// TIA Portal V17 export
// export: Created 2023-03-06T02:05:21.4493733Z, ExportSetting WithDefaults, DisplayName Totally Integrated Automation Portal, DisplayVersion V17 Update 4, DisplayName TIA Portal Openness, DisplayVersion V17 Update 4, DisplayName TIA Portal Version Control Interface, DisplayVersion V17, DisplayName STEP 7 Professional, DisplayVersion V17 Update 4, DisplayName STEP 7 Safety, DisplayVersion V17, DisplayName WinCC Professional, DisplayVersion V17 Update 4
FUNCTION "SM2_Logic" : Void   // FC70, LAD
TITLE = State Machine Logic
{ S7_Optimized_Access := 'TRUE' }
VERSION : 0.1
// stored: AutoNumber false, IsIECCheckEnabled false, SetENOAutomatically false, UDAEnableTagReadback false
   VAR_TEMP   // added for the SCL form of the ladder/FBD networks
      _w1 : Bool;
   END_VAR
BEGIN

REGION Network 1: Stop Command
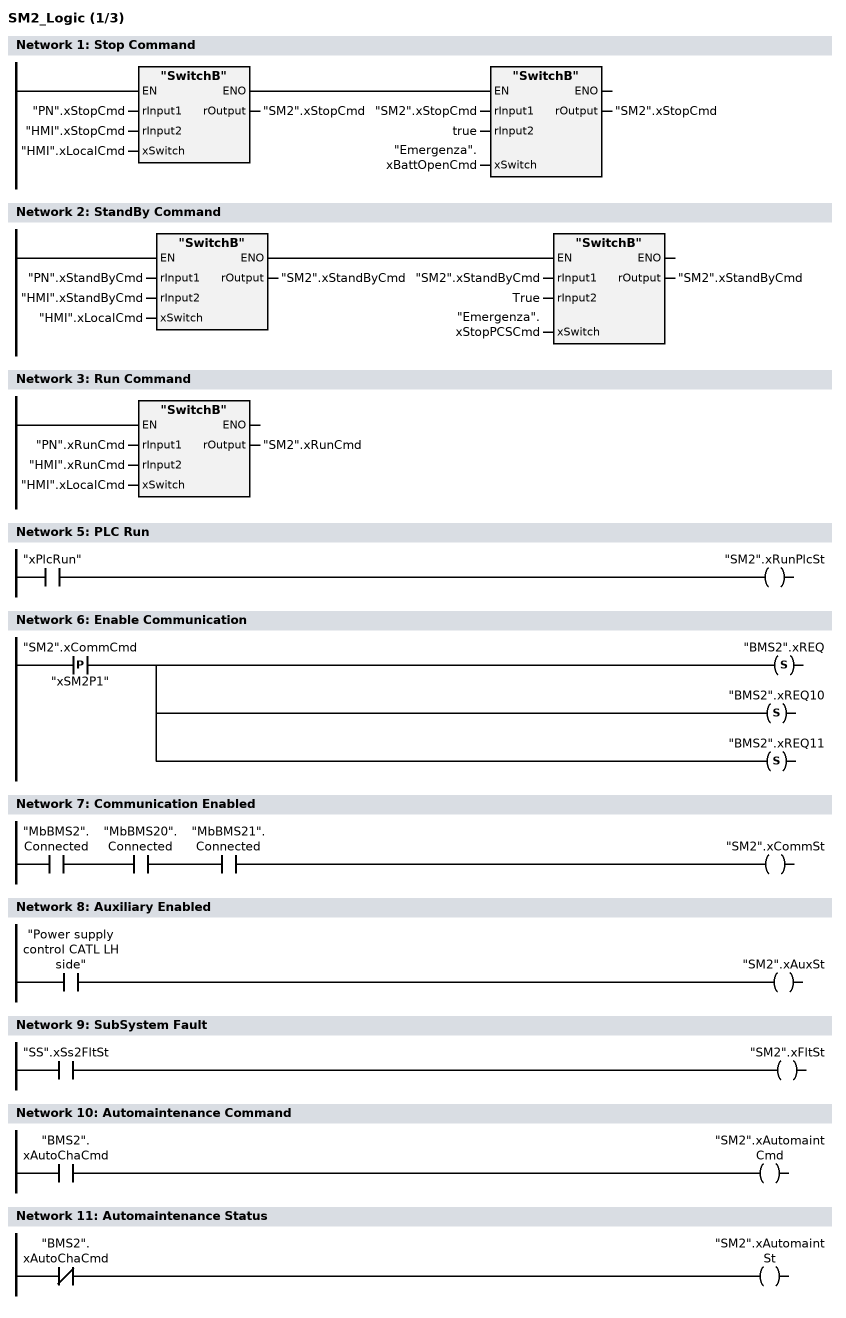
   RUNG wire#powerrail
      "SwitchB"(rInput1 := "PN".xStopCmd, rInput2 := "HMI".xStopCmd, xSwitch := "HMI".xLocalCmd, rOutput => "SM2".xStopCmd)
      "SwitchB"(rInput1 := "SM2".xStopCmd, rInput2 := true, xSwitch := "Emergenza".xBattOpenCmd, rOutput => "SM2".xStopCmd)
   END_RUNG
   // the same network as SCL:
   "SwitchB"(rInput1 := "PN".xStopCmd,
             rInput2 := "HMI".xStopCmd,
             xSwitch := "HMI".xLocalCmd,
             rOutput => "SM2".xStopCmd,
             ENO => #_w1);
   IF #_w1 THEN
       "SwitchB"(rInput1 := "SM2".xStopCmd,
                 rInput2 := true,
                 xSwitch := "Emergenza".xBattOpenCmd,
                 rOutput => "SM2".xStopCmd);
   END_IF;
END_REGION

REGION Network 2: StandBy Command
   RUNG wire#powerrail
      "SwitchB"(rInput1 := "PN".xStandByCmd, rInput2 := "HMI".xStandByCmd, xSwitch := "HMI".xLocalCmd, rOutput => "SM2".xStandByCmd)
      "SwitchB"(rInput1 := "SM2".xStandByCmd, rInput2 := True, xSwitch := "Emergenza".xStopPCSCmd, rOutput => "SM2".xStandByCmd)
   END_RUNG
   // the same network as SCL:
   "SwitchB"(rInput1 := "PN".xStandByCmd,
             rInput2 := "HMI".xStandByCmd,
             xSwitch := "HMI".xLocalCmd,
             rOutput => "SM2".xStandByCmd,
             ENO => #_w1);
   IF #_w1 THEN
       "SwitchB"(rInput1 := "SM2".xStandByCmd,
                 rInput2 := True,
                 xSwitch := "Emergenza".xStopPCSCmd,
                 rOutput => "SM2".xStandByCmd);
   END_IF;
END_REGION

REGION Network 3: Run Command
   RUNG wire#powerrail
      "SwitchB"(rInput1 := "PN".xRunCmd, rInput2 := "HMI".xRunCmd, xSwitch := "HMI".xLocalCmd, rOutput => "SM2".xRunCmd)
   END_RUNG
   // the same network as SCL:
   "SwitchB"(rInput1 := "PN".xRunCmd,
             rInput2 := "HMI".xRunCmd,
             xSwitch := "HMI".xLocalCmd,
             rOutput => "SM2".xRunCmd);
END_REGION

REGION Network 5: PLC Run
   RUNG wire#powerrail
      Contact( "xPlcRun" )
      Coil( "SM2".xRunPlcSt )
   END_RUNG
   // the same network as SCL:
   "SM2".xRunPlcSt := "xPlcRun";
END_REGION

REGION Network 6: Enable Communication
   RUNG wire#powerrail
      P_Contact(operand := "SM2".xCommCmd, bit := "xSM2P1")
      wire#w1
      S_Coil( "BMS2".xREQ )
   END_RUNG
   RUNG wire#w1
      S_Coil( "BMS2".xREQ10 )
   END_RUNG
   RUNG wire#w1
      S_Coil( "BMS2".xREQ11 )
   END_RUNG
   // the same network as SCL:
   #_w1 := "SM2".xCommCmd AND NOT "xSM2P1";   // rising edge of "SM2".xCommCmd
   "xSM2P1" := "SM2".xCommCmd;
   IF #_w1 THEN
       "BMS2".xREQ := TRUE;
       "BMS2".xREQ10 := TRUE;
       "BMS2".xREQ11 := TRUE;
   END_IF;
END_REGION

REGION Network 7: Communication Enabled
   RUNG wire#powerrail
      Contact( "MbBMS2".Connected )
      Contact( "MbBMS20".Connected )
      Contact( "MbBMS21".Connected )
      Coil( "SM2".xCommSt )
   END_RUNG
   // the same network as SCL:
   "SM2".xCommSt := "MbBMS2".Connected AND "MbBMS20".Connected AND "MbBMS21".Connected;
END_REGION

REGION Network 8: Auxiliary Enabled
   RUNG wire#powerrail
      Contact( "Power supply control CATL LH side" )
      Coil( "SM2".xAuxSt )
   END_RUNG
   // the same network as SCL:
   "SM2".xAuxSt := "Power supply control CATL LH side";
END_REGION

REGION Network 9: SubSystem Fault
   RUNG wire#powerrail
      Contact( "SS".xSs2FltSt )
      Coil( "SM2".xFltSt )
   END_RUNG
   // the same network as SCL:
   "SM2".xFltSt := "SS".xSs2FltSt;
END_REGION

REGION Network 10: Automaintenance Command
   RUNG wire#powerrail
      Contact( "BMS2".xAutoChaCmd )
      Coil( "SM2".xAutomaintCmd )
   END_RUNG
   // the same network as SCL:
   "SM2".xAutomaintCmd := "BMS2".xAutoChaCmd;
END_REGION

REGION Network 11: Automaintenance Status
   RUNG wire#powerrail
      I_Contact( "BMS2".xAutoChaCmd )
      Coil( "SM2".xAutomaintSt )
   END_RUNG
   // the same network as SCL:
   "SM2".xAutomaintSt := NOT "BMS2".xAutoChaCmd;
END_REGION

REGION Network 12: Test Command
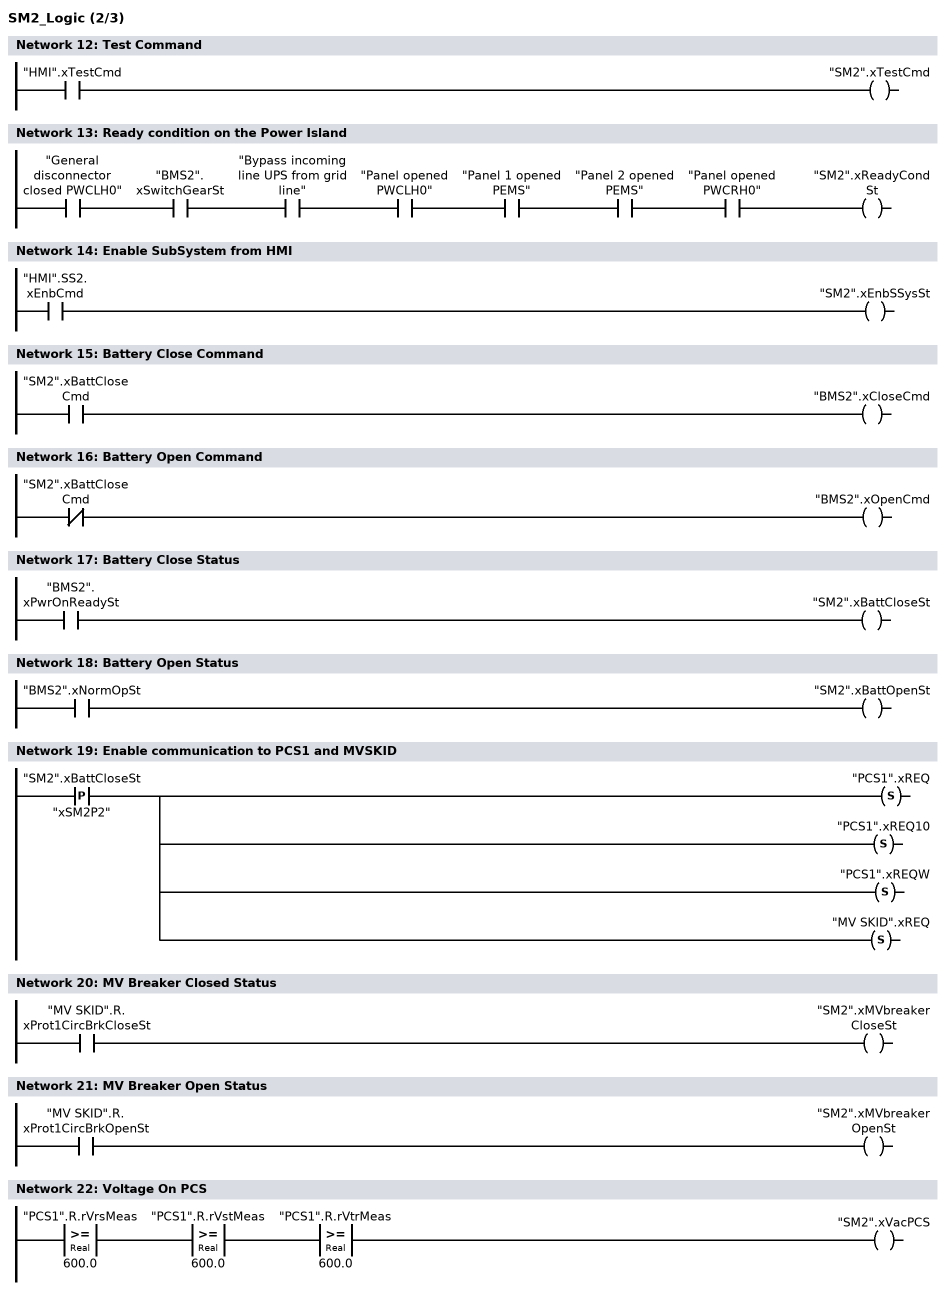
   RUNG wire#powerrail
      Contact( "HMI".xTestCmd )
      Coil( "SM2".xTestCmd )
   END_RUNG
   // the same network as SCL:
   "SM2".xTestCmd := "HMI".xTestCmd;
END_REGION

REGION Network 13: Ready condition on the Power Island
   RUNG wire#powerrail
      Contact( "General disconnector closed PWCLH0" )
      Contact( "BMS2".xSwitchGearSt )
      Contact( "Bypass incoming line UPS from grid line" )
      Contact( "Panel opened PWCLH0" )
      Contact( "Panel 1 opened PEMS" )
      Contact( "Panel 2 opened PEMS" )
      Contact( "Panel opened PWCRH0" )
      Coil( "SM2".xReadyCondSt )
   END_RUNG
   // the same network as SCL:
   "SM2".xReadyCondSt := "General disconnector closed PWCLH0" AND "BMS2".xSwitchGearSt AND "Bypass incoming line UPS from grid line" AND "Panel opened PWCLH0" AND "Panel 1 opened PEMS" AND "Panel 2 opened PEMS" AND "Panel opened PWCRH0";
END_REGION

REGION Network 14: Enable SubSystem from HMI
   RUNG wire#powerrail
      Contact( "HMI".SS2.xEnbCmd )
      Coil( "SM2".xEnbSSysSt )
   END_RUNG
   // the same network as SCL:
   "SM2".xEnbSSysSt := "HMI".SS2.xEnbCmd;
END_REGION

REGION Network 15: Battery Close Command
   RUNG wire#powerrail
      Contact( "SM2".xBattCloseCmd )
      Coil( "BMS2".xCloseCmd )
   END_RUNG
   // the same network as SCL:
   "BMS2".xCloseCmd := "SM2".xBattCloseCmd;
END_REGION

REGION Network 16: Battery Open Command
   RUNG wire#powerrail
      I_Contact( "SM2".xBattCloseCmd )
      Coil( "BMS2".xOpenCmd )
   END_RUNG
   // the same network as SCL:
   "BMS2".xOpenCmd := NOT "SM2".xBattCloseCmd;
END_REGION

REGION Network 17: Battery Close Status
   RUNG wire#powerrail
      Contact( "BMS2".xPwrOnReadySt )
      Coil( "SM2".xBattCloseSt )
   END_RUNG
   // the same network as SCL:
   "SM2".xBattCloseSt := "BMS2".xPwrOnReadySt;
END_REGION

REGION Network 18: Battery Open Status
   RUNG wire#powerrail
      Contact( "BMS2".xNormOpSt )
      Coil( "SM2".xBattOpenSt )
   END_RUNG
   // the same network as SCL:
   "SM2".xBattOpenSt := "BMS2".xNormOpSt;
END_REGION

REGION Network 19: Enable communication to PCS1 and MVSKID
   RUNG wire#powerrail
      P_Contact(operand := "SM2".xBattCloseSt, bit := "xSM2P2")
      wire#w1
      S_Coil( "PCS1".xREQ )
   END_RUNG
   RUNG wire#w1
      S_Coil( "PCS1".xREQ10 )
   END_RUNG
   RUNG wire#w1
      S_Coil( "PCS1".xREQW )
   END_RUNG
   RUNG wire#w1
      S_Coil( "MV SKID".xREQ )
   END_RUNG
   // the same network as SCL:
   #_w1 := "SM2".xBattCloseSt AND NOT "xSM2P2";   // rising edge of "SM2".xBattCloseSt
   "xSM2P2" := "SM2".xBattCloseSt;
   IF #_w1 THEN
       "PCS1".xREQ := TRUE;
       "PCS1".xREQ10 := TRUE;
       "PCS1".xREQW := TRUE;
       "MV SKID".xREQ := TRUE;
   END_IF;
END_REGION

REGION Network 20: MV Breaker Closed Status
   RUNG wire#powerrail
      Contact( "MV SKID".R.xProt1CircBrkCloseSt )
      Coil( "SM2".xMVbreakerCloseSt )
   END_RUNG
   // the same network as SCL:
   "SM2".xMVbreakerCloseSt := "MV SKID".R.xProt1CircBrkCloseSt;
END_REGION

REGION Network 21: MV Breaker Open Status
   RUNG wire#powerrail
      Contact( "MV SKID".R.xProt1CircBrkOpenSt )
      Coil( "SM2".xMVbreakerOpenSt )
   END_RUNG
   // the same network as SCL:
   "SM2".xMVbreakerOpenSt := "MV SKID".R.xProt1CircBrkOpenSt;
END_REGION

REGION Network 22: Voltage On PCS
   RUNG wire#powerrail
      { S7_Templates := "SrcType := Real" } GE_Contact(in1 := "PCS1".R.rVrsMeas, in2 := 600.0)
      { S7_Templates := "SrcType := Real" } GE_Contact(in1 := "PCS1".R.rVstMeas, in2 := 600.0)
      { S7_Templates := "SrcType := Real" } GE_Contact(in1 := "PCS1".R.rVtrMeas, in2 := 600.0)
      Coil( "SM2".xVacPCS )
   END_RUNG
   // the same network as SCL:
   "SM2".xVacPCS := ("PCS1".R.rVrsMeas >= 600.0) AND ("PCS1".R.rVstMeas >= 600.0) AND ("PCS1".R.rVtrMeas >= 600.0);
END_REGION

REGION Network 23: PCS Ready Status
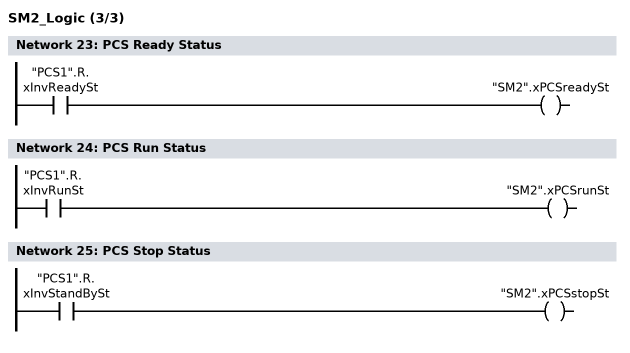
   RUNG wire#powerrail
      Contact( "PCS1".R.xInvReadySt )
      Coil( "SM2".xPCSreadySt )
   END_RUNG
   // the same network as SCL:
   "SM2".xPCSreadySt := "PCS1".R.xInvReadySt;
END_REGION

REGION Network 24: PCS Run Status
   RUNG wire#powerrail
      Contact( "PCS1".R.xInvRunSt )
      Coil( "SM2".xPCSrunSt )
   END_RUNG
   // the same network as SCL:
   "SM2".xPCSrunSt := "PCS1".R.xInvRunSt;
END_REGION

REGION Network 25: PCS Stop Status
   RUNG wire#powerrail
      Contact( "PCS1".R.xInvStandBySt )
      Coil( "SM2".xPCSstopSt )
   END_RUNG
   // the same network as SCL:
   "SM2".xPCSstopSt := "PCS1".R.xInvStandBySt;
END_REGION
END_FUNCTION
